// TIA Portal V18 export
// export: Created 2025-12-01T12:38:48.7770701Z, ExportSetting None, DisplayName Totally Integrated Automation Portal, DisplayVersion V18 Update 5, DisplayName TIA Portal Openness, DisplayVersion V18 Update 5, DisplayName TIA Portal Teamcenter Gateway, DisplayVersion V18, DisplayName TIA Portal Version Control Interface, DisplayVersion V18, DisplayName STEP 7 Professional, DisplayVersion V18 Update 5, DisplayName STEP 7 Safety, DisplayVersion V18, DisplayName WinCC Professional, DisplayVersion V18 Update 5
FUNCTION_BLOCK "ST10_FB_S7connect"   // FB900, LAD
{ S7_Optimized_Access := 'TRUE' }
// stored: AutoNumber false, MemoryReserve 100, SetENOAutomatically false
   VAR_INPUT
      "CLOCK_0.2_SEC" : Bool;
   END_VAR
   VAR
      Always_On : Bool;
      Status_Get : Array[1..6] of Struct
         NDR : Bool;
         Error : Bool;
         Status : Int;
      END_STRUCT;
      Status_Put : Array[1..6] of Struct
         Done : Bool;
         Error : Bool;
         Status : Int;
      END_STRUCT;
      GET_Instance1 { S7_SetPoint := 'True'} : GET;
      GET_Instance2 { S7_SetPoint := 'True'} : GET;
      PUT_Instance1 { S7_SetPoint := 'True'} : PUT;
      PUT_Instance2 { S7_SetPoint := 'True'} : PUT;
      PLs { S7_SetPoint := 'True'} : Array[1..6] of Bool;
   END_VAR
   VAR DB_SPECIFIC
      TON : Array[1..5] of TON_TIME;
   END_VAR
   VAR
      NextStation_OffLine : Bool;   // S7心跳超时
   END_VAR
BEGIN

REGION Network 1: **************** 和40交互 **************** / **************** ****************
END_REGION

REGION Network 2: PUT
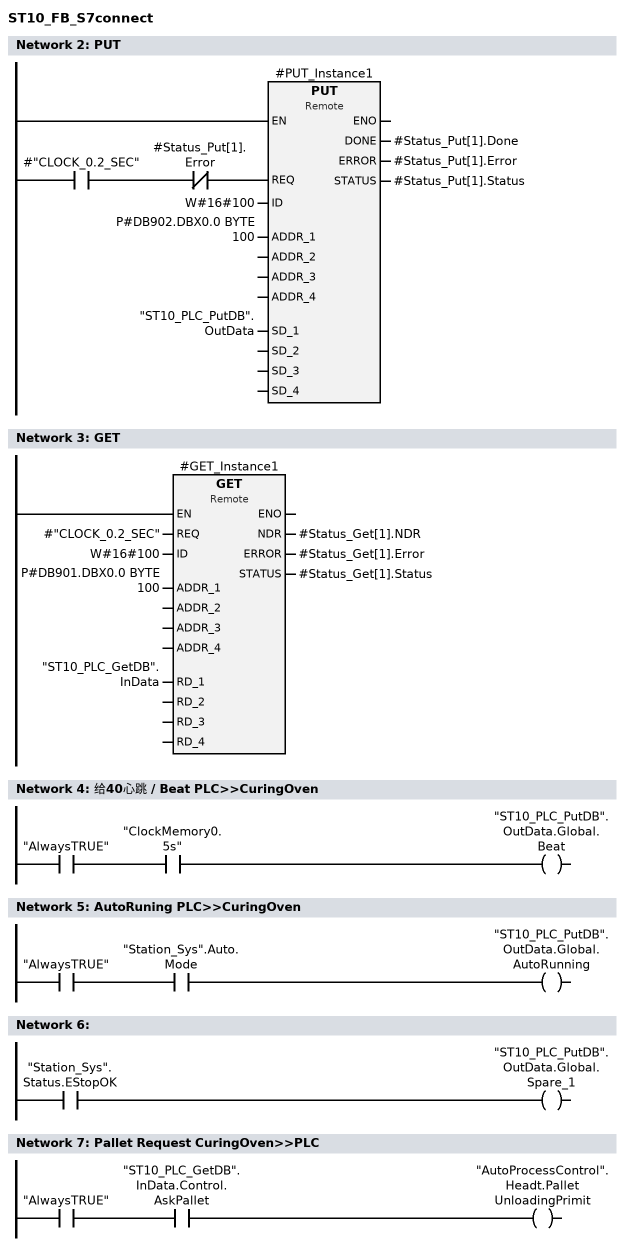
   RUNG wire#powerrail
      { S7_Templates := "[remote_type := Remote, local_type := Variant]" } #PUT_Instance1.PUT(REQ := wire#w1, ID := W#16#100, ADDR_1 := P#DB902.DBX0.0 BYTE 100, ADDR_2 :=, ADDR_3 :=, ADDR_4 :=, SD_1 := "ST10_PLC_PutDB".OutData, SD_2 :=, SD_3 :=, SD_4 :=, DONE => #Status_Put[1].Done, ERROR => #Status_Put[1].Error, STATUS => #Status_Put[1].Status)
   END_RUNG
   RUNG wire#powerrail
      Contact( #"CLOCK_0.2_SEC" )
      I_Contact( #Status_Put[1].Error )
   END_RUNG wire#w1
   // the same network as SCL:
   #PUT_Instance1(REQ := #"CLOCK_0.2_SEC" AND NOT #Status_Put[1].Error,   // PUT
                  ID := W#16#100,
                  ADDR_1 := P#DB902.DBX0.0 BYTE 100,
                  SD_1 := "ST10_PLC_PutDB".OutData,
                  DONE => #Status_Put[1].Done,
                  ERROR => #Status_Put[1].Error,
                  STATUS => #Status_Put[1].Status);
END_REGION

REGION Network 3: GET
   RUNG wire#powerrail
      { S7_Templates := "[remote_type := Remote, local_type := Variant]" } #GET_Instance1.GET(REQ := #"CLOCK_0.2_SEC", ID := W#16#100, ADDR_1 := P#DB901.DBX0.0 BYTE 100, ADDR_2 :=, ADDR_3 :=, ADDR_4 :=, RD_1 := "ST10_PLC_GetDB".InData, RD_2 :=, RD_3 :=, RD_4 :=, NDR => #Status_Get[1].NDR, ERROR => #Status_Get[1].Error, STATUS => #Status_Get[1].Status)
   END_RUNG
   // the same network as SCL:
   #GET_Instance1(REQ := #"CLOCK_0.2_SEC",   // GET
                  ID := W#16#100,
                  ADDR_1 := P#DB901.DBX0.0 BYTE 100,
                  RD_1 := "ST10_PLC_GetDB".InData,
                  NDR => #Status_Get[1].NDR,
                  ERROR => #Status_Get[1].Error,
                  STATUS => #Status_Get[1].Status);
END_REGION

REGION Network 4: 给40心跳 / Beat PLC>>CuringOven
   RUNG wire#powerrail
      Contact( "AlwaysTRUE" )
      Contact( "ClockMemory0.5s" )
      Coil( "ST10_PLC_PutDB".OutData.Global.Beat )
   END_RUNG
   // the same network as SCL:
   "ST10_PLC_PutDB".OutData.Global.Beat := "AlwaysTRUE" AND "ClockMemory0.5s";
END_REGION

REGION Network 5: AutoRuning PLC>>CuringOven
   RUNG wire#powerrail
      Contact( "AlwaysTRUE" )
      Contact( "Station_Sys".Auto.Mode )
      Coil( "ST10_PLC_PutDB".OutData.Global.AutoRunning )
   END_RUNG
   // the same network as SCL:
   "ST10_PLC_PutDB".OutData.Global.AutoRunning := "AlwaysTRUE" AND "Station_Sys".Auto.Mode;
END_REGION

REGION Network 6
   RUNG wire#powerrail
      Contact( "Station_Sys".Status.EStopOK )
      Coil( "ST10_PLC_PutDB".OutData.Global.Spare_1 )
   END_RUNG
   // the same network as SCL:
   "ST10_PLC_PutDB".OutData.Global.Spare_1 := "Station_Sys".Status.EStopOK;
END_REGION

REGION Network 7: Pallet Request CuringOven>>PLC
   RUNG wire#powerrail
      Contact( "AlwaysTRUE" )
      Contact( "ST10_PLC_GetDB".InData.Control.AskPallet )
      Coil( "AutoProcessControl".Headt.PalletUnloadingPrimit )
   END_RUNG
   // the same network as SCL:
   "AutoProcessControl".Headt.PalletUnloadingPrimit := "AlwaysTRUE" AND "ST10_PLC_GetDB".InData.Control.AskPallet;
END_REGION
END_FUNCTION_BLOCK
